TYPE ST_KeyenceLaser_Edit_Request :
STRUCT
Edit_Start_Request			: BIT;
Reserve_0					: BIT;
Reserve_1					: BIT;
Reserve_2					: BIT;
Reserve_3					: BIT;
Reserve_4					: BIT;
Reserve_5					: BIT;
Reserve_6					: BIT;
END_STRUCT
END_TYPE

(* stored: Version 1.1.0.1, ProductVersion 3.1.4024.11
   DUT ST_KeyenceLaser_Edit_Request: Id {e3b51200-645c-4fbe-819f-161d911e3c0f} *)
